# EPICS autosave request: iocs/tlbc2IOC/iocBoot/ioctlbc2/ioc.req
file "ADTLBC2_settings.req", P=$(P), R=cam1:
file "plugins.req",          P=$(P)
